Fanuc KAREL source: kb00013.KL

-- PROVISIONAL review KL for V940-1; original PC SHA256 ba460e5a32155135fb6223ae8b66ccdcffbb4b78bcee7e253fa9da5b918012d5
-- Incomplete behavior may be omitted. Consult companion uncertainty JSON. Do not deploy.
PROGRAM KB00013
%NOLOCKGROUP
BEGIN
  -- V9_ZERO_TABLE_METADATA_HINT layout=0002_ascii; no indexed target words; source/name/runtime held
  -- UNRESOLVED_PC offsets 5-12; opcodes 9D,23
  -- UNRESOLVED_PC offsets 17-24; opcodes 9D,23
  -- UNRESOLVED_PC offsets 29-51; opcodes 27,22,22,22,31
  -- UNRESOLVED_PC offsets 56-60; opcodes 7F
END KB00013
